{attribute 'qualified_only'}
{attribute 'strict'}

//-----------------------------------------------------------------------------------------
//
//                  				ENUM_CNC_Type
//
//							Enumération des types CNC			
//-----------------------------------------------------------------------------------------
//
//Auteur: G.GOETZ
//Création: 27.01.2026
//Dernière modification : 27.01.2026 (G.GOETZ)
//       			
//-----------------------------------------------------------------------------------------
//
//     							Liste des modifications  	
//
// 27.01.2026 (G.GOETZ) -> Création		
//-----------------------------------------------------------------------------------------

TYPE ENUM_CNC_Type :
(
	(*Unknow := 0 , // Unknow type*)
	Fanuc := 1 , // Fanuc CNC type
	Heidenhain := 2 // Heidenhain CNC type
);
END_TYPE

(* stored: Version 1.1.0.1, ProductVersion 3.1.4024.13
   DUT ENUM_CNC_Type: Id {49122184-1ded-43ce-a2c7-a17124c283bc} *)
